{attribute addProperty BoxType "EL1259-0000-0017"}
{attribute addProperty Id "CtrlAT %Q*Ctrl_8EDFA0AF607.51OutputsAT %Q*Outputs_C23F921918623.2533Output_event_timeAT %Q*ARRAY[0 ..9] OF UDINT320400"}
{attribute addProperty CRC "3926941601"}
{attribute addProperty SizeInBites "566"}
{attribute addProperty SizeInBytes "70.75"}
TYPE MTO_Outputs_10x_Channel_24D255B1 :
STRUCT
	{attribute addProperty Name "Ctrl"}
	Ctrl AT %Q* : Ctrl_8EDFA0AF;
	{attribute addProperty Name "Outputs"}
	Outputs AT %Q* : Outputs_C23F9219;
	{attribute addProperty Name "Output_event_time"}
	Output_event_time AT %Q* : ARRAY[0 ..9] OF UDINT;
END_STRUCT
END_TYPE

(* stored: Version 1.2.0.0, ProductVersion 3.1.4024.9
   DUT MTO_Outputs_10x_Channel_24D255B1: Id {3989e780-6cce-4e11-baa2-eb9bea0f6ef2} *)
